(* IEC 61131-3 sources: Industry-PLC-LLM/data/PLCBEAD_repo/PLCBEAD_PLCEmbed-main/PLC-BEAD/Source/GEB/BYTE_TO_STRB, 1 file *)

(* ---- BYTE_TO_STRB.ST ---- *)
FUNCTION_BLOCK BYTE_TO_STRB_Block
	VAR_INPUT
		IN :	BYTE;
	END_VAR

	VAR_OUTPUT
		BYTE_TO_STRB :	STRING;
	END_VAR

	VAR
		i :	INT;
		IN_P : BYTE;
	END_VAR
	IN_P := IN;
	BYTE_TO_STRB := '';
	FOR i := 1 TO 8 DO
		IF (IN_P AND BYTE#2#1000_0000) = BYTE#2#1000_0000 THEN
			BYTE_TO_STRB := CONCAT(BYTE_TO_STRB,'1');
		ELSE
			BYTE_TO_STRB := CONCAT(BYTE_TO_STRB,'0');
		END_IF;
		IN_P := SHL(IN_P, 1);
	END_FOR;

END_FUNCTION_BLOCK

PROGRAM program0
  VAR
    LocalVar0 : BYTE;
	LocalOUT  : STRING;
	func_block : BYTE_TO_STRB_Block;
  END_VAR
	func_block.IN  := LocalVar0;
	func_block();
	LocalOUT := func_block.BYTE_TO_STRB;

END_PROGRAM
